TYPE stStationInfo :
STRUCT
	Clear : BOOL;
	Complete : BOOL;
	Operating : BOOL;
	Ready : BOOL;
	HasMover : BOOL;
END_STRUCT
END_TYPE

(* stored: Version 1.1.0.1, ProductVersion 3.1.4024.11
   DUT stStationInfo: Id {533a335d-24db-4b41-ade9-236dde69feb4} *)
